   Y[2027] := 0.748582;
   Y[2028] := 0.7531839;
   Y[2029] := 0.7531839;
   Y[2030] := 0.75165;
   Y[2031] := 0.7531839;
   Y[2032] := 0.750116;
   Y[2033] := 0.7547179;
   Y[2034] := 0.748582;
   Y[2035] := 0.7593198;
   Y[2036] := 0.750116;
   Y[2037] := 0.7577859;
   Y[2038] := 0.7531839;
   Y[2039] := 0.7531839;
   Y[2040] := 0.745514;
   Y[2041] := 0.7639218;
   Y[2042] := 0.748582;
   Y[2043] := 0.7623878;
   Y[2044] := 0.750116;
   Y[2045] := 0.7577859;
   Y[2046] := 0.747048;
   Y[2047] := 0.7623878;
   Y[2048] := 0.748582;
   Y[2049] := 0.7700577;
   Y[2050] := 0.7424461;
   Y[2051] := 0.7608538;
   Y[2052] := 0.7531839;
   Y[2053] := 0.7577859;
   Y[2054] := 0.7531839;
   Y[2055] := 0.7577859;
   Y[2056] := 0.7577859;
   Y[2057] := 0.7531839;
   Y[2058] := 0.7593198;
   Y[2059] := 0.7531839;
   Y[2060] := 0.7623878;
   Y[2061] := 0.750116;
   Y[2062] := 0.7623878;
   Y[2063] := 0.7531839;
   Y[2064] := 0.7623878;
   Y[2065] := 0.750116;
   Y[2066] := 0.7654558;
   Y[2067] := 0.7562519;
   Y[2068] := 0.7577859;
   Y[2069] := 0.750116;
   Y[2070] := 0.7669898;
   Y[2071] := 0.747048;
   Y[2072] := 0.7669898;
   Y[2073] := 0.748582;
   Y[2074] := 0.7731256;
   Y[2075] := 0.747048;
   Y[2076] := 0.7654558;
   Y[2077] := 0.748582;
   Y[2078] := 0.7654558;
   Y[2079] := 0.750116;
   Y[2080] := 0.7608538;
   Y[2081] := 0.7547179;
   Y[2082] := 0.7562519;
   Y[2083] := 0.7562519;
   Y[2084] := 0.75165;
   Y[2085] := 0.7562519;
   Y[2086] := 0.7439801;
   Y[2087] := 0.7378441;
   Y[2088] := 0.7056305;
   Y[2089] := 0.6626791;
   Y[2090] := 0.5798442;
   Y[2091] := 0.523087;
   Y[2092] := 0.4617278;
   Y[2093] := 0.4203104;
   Y[2094] := 0.4003687;
   Y[2095] := 0.3926988;
   Y[2096] := 0.374291;
   Y[2097] := 0.3666211;
   Y[2098] := 0.3620192;
   Y[2099] := 0.3574172;
   Y[2100] := 0.3589512;
   Y[2101] := 0.3620192;
   Y[2102] := 0.3666211;
   Y[2103] := 0.3681551;
   Y[2104] := 0.3635531;
   Y[2105] := 0.3574172;
   Y[2106] := 0.3604852;
   Y[2107] := 0.3497473;
   Y[2108] := 0.3574172;
   Y[2109] := 0.3512813;
   Y[2110] := 0.3512813;
   Y[2111] := 0.3620192;
   Y[2112] := 0.3574172;
   Y[2113] := 0.3482133;
   Y[2114] := 0.3482133;
   Y[2115] := 0.3543493;
   Y[2116] := 0.3451454;
   Y[2117] := 0.3543493;
   Y[2118] := 0.3405434;
   Y[2119] := 0.3543493;
   Y[2120] := 0.3451454;
   Y[2121] := 0.3558832;
   Y[2122] := 0.3451454;
   Y[2123] := 0.3558832;
   Y[2124] := 0.3482133;
   Y[2125] := 0.3604852;
   Y[2126] := 0.3666211;
   Y[2127] := 0.3558832;
   Y[2128] := 0.3650871;
   Y[2129] := 0.3589512;
   Y[2130] := 0.3620192;
   Y[2131] := 0.3466794;
   Y[2132] := 0.3497473;
   Y[2133] := 0.3574172;
   Y[2134] := 0.3589512;
   Y[2135] := 0.369689;
   Y[2136] := 0.3635531;
   Y[2137] := 0.3788929;
   Y[2138] := 0.369689;
   Y[2139] := 0.3773589;
   Y[2140] := 0.372757;
   Y[2141] := 0.371223;
   Y[2142] := 0.3819609;
   Y[2143] := 0.375825;
   Y[2144] := 0.3773589;
   Y[2145] := 0.372757;
   Y[2146] := 0.3911648;
   Y[2147] := 0.3880968;
   Y[2148] := 0.371223;
   Y[2149] := 0.374291;
   Y[2150] := 0.374291;
   Y[2151] := 0.374291;
   Y[2152] := 0.374291;
   Y[2153] := 0.3681551;
   Y[2154] := 0.3788929;
   Y[2155] := 0.3804269;
   Y[2156] := 0.3834949;
   Y[2157] := 0.3865628;
   Y[2158] := 0.3926988;
   Y[2159] := 0.3926988;
   Y[2160] := 0.3865628;
   Y[2161] := 0.3942327;
   Y[2162] := 0.3804269;
   Y[2163] := 0.3911648;
   Y[2164] := 0.3880968;
   Y[2165] := 0.3880968;
   Y[2166] := 0.3865628;
   Y[2167] := 0.3988347;
   Y[2168] := 0.3942327;
   Y[2169] := 0.3819609;
   Y[2170] := 0.3911648;
   Y[2171] := 0.3988347;
   Y[2172] := 0.3911648;
   Y[2173] := 0.3850288;
   Y[2174] := 0.4003687;
   Y[2175] := 0.3926988;
   Y[2176] := 0.3896308;
   Y[2177] := 0.369689;
   Y[2178] := 0.3788929;
   Y[2179] := 0.3834949;
   Y[2180] := 0.3973007;
   Y[2181] := 0.3850288;
   Y[2182] := 0.3957667;
   Y[2183] := 0.3911648;
   Y[2184] := 0.4049706;
   Y[2185] := 0.3957667;
   Y[2186] := 0.4111065;
   Y[2187] := 0.4126405;
   Y[2188] := 0.4049706;
   Y[2189] := 0.4034366;
   Y[2190] := 0.4157085;
   Y[2191] := 0.4187764;
   Y[2192] := 0.4126405;
   Y[2193] := 0.4203104;
   Y[2194] := 0.4187764;
   Y[2195] := 0.4264463;
   Y[2196] := 0.4095725;
   Y[2197] := 0.4279803;
   Y[2198] := 0.4172424;
   Y[2199] := 0.4325822;
   Y[2200] := 0.4141745;
   Y[2201] := 0.4341162;
   Y[2202] := 0.4325822;
   Y[2203] := 0.4325822;
   Y[2204] := 0.4233783;
   Y[2205] := 0.4295143;
   Y[2206] := 0.4448541;
   Y[2207] := 0.4295143;
   Y[2208] := 0.4264463;
   Y[2209] := 0.4249123;
   Y[2210] := 0.4371842;
   Y[2211] := 0.4203104;
   Y[2212] := 0.4233783;
   Y[2213] := 0.4249123;
   Y[2214] := 0.4264463;
   Y[2215] := 0.4141745;
   Y[2216] := 0.4187764;
   Y[2217] := 0.4295143;
   Y[2218] := 0.4295143;
   Y[2219] := 0.4203104;
   Y[2220] := 0.4264463;
   Y[2221] := 0.4249123;
   Y[2222] := 0.4203104;
   Y[2223] := 0.4111065;
   Y[2224] := 0.4157085;
   Y[2225] := 0.4264463;
   Y[2226] := 0.4065046;
   Y[2227] := 0.4141745;
   Y[2228] := 0.4218444;
   Y[2229] := 0.4310482;
   Y[2230] := 0.4187764;
   Y[2231] := 0.4218444;
   Y[2232] := 0.4264463;
   Y[2233] := 0.4233783;
   Y[2234] := 0.4203104;
   Y[2235] := 0.4310482;
   Y[2236] := 0.4341162;
   Y[2237] := 0.4203104;
   Y[2238] := 0.4187764;
   Y[2239] := 0.4218444;
   Y[2240] := 0.4295143;
   Y[2241] := 0.4141745;
   Y[2242] := 0.4203104;
   Y[2243] := 0.4203104;
   Y[2244] := 0.4233783;
   Y[2245] := 0.4126405;
   Y[2246] := 0.4233783;
   Y[2247] := 0.4310482;
   Y[2248] := 0.4279803;
   Y[2249] := 0.4279803;
   Y[2250] := 0.4295143;
   Y[2251] := 0.4310482;
   Y[2252] := 0.4249123;
   Y[2253] := 0.4264463;
   Y[2254] := 0.4295143;
   Y[2255] := 0.4264463;
   Y[2256] := 0.4264463;
   Y[2257] := 0.4341162;
   Y[2258] := 0.4356502;
   Y[2259] := 0.4325822;
   Y[2260] := 0.4402521;
   Y[2261] := 0.4571259;
   Y[2262] := 0.4540579;
   Y[2263] := 0.4387181;
   Y[2264] := 0.4540579;
   Y[2265] := 0.4632618;
   Y[2266] := 0.4571259;
   Y[2267] := 0.446388;
   Y[2268] := 0.4525239;
   Y[2269] := 0.4402521;
   Y[2270] := 0.4402521;
   Y[2271] := 0.4371842;
   Y[2272] := 0.4555919;
   Y[2273] := 0.4387181;
   Y[2274] := 0.4433201;
   Y[2275] := 0.4448541;
   Y[2276] := 0.4555919;
   Y[2277] := 0.4371842;
   Y[2278] := 0.4448541;
   Y[2279] := 0.449456;
   Y[2280] := 0.4433201;
   Y[2281] := 0.4325822;
   Y[2282] := 0.4371842;
   Y[2283] := 0.4356502;
   Y[2284] := 0.4187764;
   Y[2285] := 0.4203104;
   Y[2286] := 0.4187764;
   Y[2287] := 0.4095725;
   Y[2288] := 0.4126405;
   Y[2289] := 0.4233783;
   Y[2290] := 0.4279803;
   Y[2291] := 0.4157085;
   Y[2292] := 0.4080386;
   Y[2293] := 0.3957667;
   Y[2294] := 0.4003687;
   Y[2295] := 0.3773589;
   Y[2296] := 0.374291;
   Y[2297] := 0.3896308;
   Y[2298] := 0.3880968;
   Y[2299] := 0.3804269;
   Y[2300] := 0.371223;
   Y[2301] := 0.3788929;
   Y[2302] := 0.3804269;
   Y[2303] := 0.3451454;
   Y[2304] := 0.3604852;
   Y[2305] := 0.3650871;
   Y[2306] := 0.3589512;
   Y[2307] := 0.3390095;
   Y[2308] := 0.3267376;
   Y[2309] := 0.3451454;
   Y[2310] := 0.3344075;
   Y[2311] := 0.3374755;
   Y[2312] := 0.3083299;
   Y[2313] := 0.2883881;
   Y[2314] := 0.2899221;
   Y[2315] := 0.2807182;
   Y[2316] := 0.2822522;
   Y[2317] := 0.2669124;
   Y[2318] := 0.2607765;
   Y[2319] := 0.2500387;
   Y[2320] := 0.2515726;
   Y[2321] := 0.2454367;
   Y[2322] := 0.2715144;
   Y[2323] := 0.2653784;
   Y[2324] := 0.2377668;
   Y[2325] := 0.228563;
   Y[2326] := 0.2393008;
   Y[2327] := 0.2592425;
   Y[2328] := 0.2669124;
   Y[2329] := 0.2899221;
   Y[2330] := 0.2745823;
   Y[2331] := 0.2592425;
   Y[2332] := 0.2883881;
   Y[2333] := 0.2715144;
   Y[2334] := 0.2761163;
   Y[2335] := 0.2745823;
   Y[2336] := 0.2653784;
   Y[2337] := 0.2577085;
   Y[2338] := 0.2546406;
   Y[2339] := 0.2454367;
   Y[2340] := 0.2439027;
   Y[2341] := 0.2423688;
   Y[2342] := 0.2377668;
   Y[2343] := 0.2316309;
   Y[2344] := 0.220893;
   Y[2345] := 0.2178251;
   Y[2346] := 0.2132231;
   Y[2347] := 0.2147571;
   Y[2348] := 0.2086212;
   Y[2349] := 0.2086212;
   Y[2350] := 0.1994173;
   Y[2351] := 0.1917474;
   Y[2352] := 0.1902135;
   Y[2353] := 0.1856115;
   Y[2354] := 0.1810096;
   Y[2355] := 0.1810096;
   Y[2356] := 0.1794756;
   Y[2357] := 0.1764076;
   Y[2358] := 0.1718057;
   Y[2359] := 0.1656698;
   Y[2360] := 0.1610678;
   Y[2361] := 0.1579999;
   Y[2362] := 0.1564659;
   Y[2363] := 0.15033;
   Y[2364] := 0.148796;
   Y[2365] := 0.148796;
   Y[2366] := 0.147262;
   Y[2367] := 0.1457281;
   Y[2368] := 0.1411261;
   Y[2369] := 0.1380582;
   Y[2370] := 0.1334562;
   Y[2371] := 0.1303883;
   Y[2372] := 0.1273203;
   Y[2373] := 0.1257863;
   Y[2374] := 0.1211844;
   Y[2375] := 0.1196504;
   Y[2376] := 0.1181164;
   Y[2377] := 0.1181164;
   Y[2378] := 0.1165824;
   Y[2379] := 0.1150485;
   Y[2380] := 0.1135145;
   Y[2381] := 0.1089125;
   Y[2382] := 0.1073786;
   Y[2383] := 0.1043106;
   Y[2384] := 0.1012426;
   Y[2385] := 0.1012426;
   Y[2386] := 0.09664071;
   Y[2387] := 0.09664071;
   Y[2388] := 0.09357275;
   Y[2389] := 0.09357275;
   Y[2390] := 0.09050479;
   Y[2391] := 0.08897081;
   Y[2392] := 0.08897081;
   Y[2393] := 0.08897081;
   Y[2394] := 0.08743683;
   Y[2395] := 0.08743683;
   Y[2396] := 0.08436887;
   Y[2397] := 0.08283489;
   Y[2398] := 0.08130091;
   Y[2399] := 0.07976694;
   Y[2400] := 0.07823295;
   Y[2401] := 0.075165;
   Y[2402] := 0.07363102;
   Y[2403] := 0.07363102;
   Y[2404] := 0.07209703;
   Y[2405] := 0.07056306;
   Y[2406] := 0.06902908;
   Y[2407] := 0.06902908;
   Y[2408] := 0.0674951;
   Y[2409] := 0.06596112;
   Y[2410] := 0.06596112;
   Y[2411] := 0.06289316;
   Y[2412] := 0.06442714;
   Y[2413] := 0.06289316;
   Y[2414] := 0.06289316;
   Y[2415] := 0.06135918;
   Y[2416] := 0.06135918;
   Y[2417] := 0.06135918;
   Y[2418] := 0.0598252;
   Y[2419] := 0.0598252;
   Y[2420] := 0.0598252;
   Y[2421] := 0.05829122;
   Y[2422] := 0.05675724;
   Y[2423] := 0.05522326;
   Y[2424] := 0.05368928;
   Y[2425] := 0.0521553;
   Y[2426] := 0.0521553;
   Y[2427] := 0.05062132;
   Y[2428] := 0.05062132;
   Y[2429] := 0.05062132;
   Y[2430] := 0.05062132;
   Y[2431] := 0.04755336;
   Y[2432] := 0.04908735;
   Y[2433] := 0.04601939;
   Y[2434] := 0.04755336;
   Y[2435] := 0.04601939;
   Y[2436] := 0.04601939;
   Y[2437] := 0.04601939;
   Y[2438] := 0.04295143;
   Y[2439] := 0.04295143;
   Y[2440] := 0.04295143;
   Y[2441] := 0.04141745;
   Y[2442] := 0.04141745;
   Y[2443] := 0.04141745;
   Y[2444] := 0.04295143;
   Y[2445] := 0.04141745;
   Y[2446] := 0.04141745;
   Y[2447] := 0.03988347;
   Y[2448] := 0.03988347;
   Y[2449] := 0.03988347;
   Y[2450] := 0.04141745;
   Y[2451] := 0.03988347;
   Y[2452] := 0.03988347;
   Y[2453] := 0.03988347;
   Y[2454] := 0.03988347;
   Y[2455] := 0.03834949;
   Y[2456] := 0.03988347;
   Y[2457] := 0.03681551;
   Y[2458] := 0.03681551;
   Y[2459] := 0.03681551;
   Y[2460] := 0.03374755;
   Y[2461] := 0.03528153;
   Y[2462] := 0.03374755;
   Y[2463] := 0.03221357;
   Y[2464] := 0.03374755;
   Y[2465] := 0.03374755;
   Y[2466] := 0.03221357;
   Y[2467] := 0.03528153;
   Y[2468] := 0.03374755;
   Y[2469] := 0.03221357;
   Y[2470] := 0.03374755;
   Y[2471] := 0.03221357;
   Y[2472] := 0.03374755;
   Y[2473] := 0.03221357;
   Y[2474] := 0.03221357;
   Y[2475] := 0.03221357;
   Y[2476] := 0.03221357;
   Y[2477] := 0.03221357;
   Y[2478] := 0.03067959;
   Y[2479] := 0.03067959;
   Y[2480] := 0.03067959;
   Y[2481] := 0.02914561;
   Y[2482] := 0.02914561;
   Y[2483] := 0.02761163;
   Y[2484] := 0.02914561;
   Y[2485] := 0.02607765;
   Y[2486] := 0.02761163;
   Y[2487] := 0.02761163;
   Y[2488] := 0.02761163;
   Y[2489] := 0.02761163;
   Y[2490] := 0.02761163;
   Y[2491] := 0.02914561;
   Y[2492] := 0.02761163;
   Y[2493] := 0.02914561;
   Y[2494] := 0.02761163;
   Y[2495] := 0.02761163;
   Y[2496] := 0.02761163;
   Y[2497] := 0.02607765;
   Y[2498] := 0.02914561;
   Y[2499] := 0.02761163;

END_DATA_BLOCK

FUNCTION "VecDivVal" : Void
{ S7_Optimized_Access := 'TRUE' }
VERSION : 0.1
   VAR_INPUT
      A : Array[0.."n"] of Real;
      val : Real;
   END_VAR

   VAR_OUTPUT
      C : Array[0.."n"] of Real;
   END_VAR

   VAR_TEMP
      i : DInt;
      j : DInt;
   END_VAR


BEGIN
	FOR #i := 0 TO "n" DO
	    #C[#i] := #A[#i] / #val;
	END_FOR;

END_FUNCTION

FUNCTION "MulVecRowVecCol" : Void
{ S7_Optimized_Access := 'TRUE' }
VERSION : 0.1
   VAR_INPUT
      A : Array[0.."n"] of Real;
      B : Array[0.."n"] of Real;
   END_VAR

   VAR_OUTPUT
      s : Real;
   END_VAR

   VAR_TEMP
      i : DInt;
   END_VAR


BEGIN
	#s := 0.0;
	FOR #i := 0 TO "n" DO
	    #s := #s + #A[#i] * #B[#i];
	END_FOR;

END_FUNCTION

FUNCTION "MulVecColVecRow" : Void
{ S7_Optimized_Access := 'TRUE' }
VERSION : 0.1
   VAR_INPUT
      A : Array[0.."n"] of Real;
      B : Array[0.."n"] of Real;
   END_VAR

   VAR_OUTPUT
      C : Array[0.."n", 0.."n"] of Real;
   END_VAR

   VAR_TEMP
      i : DInt;
      j : DInt;
   END_VAR


BEGIN
	FOR #i := 0 TO "n" DO
	    FOR #j := 0 TO "n" DO
	        #C[#i, #j] := #A[#i] * #B[#j];
	    END_FOR;
	END_FOR;

END_FUNCTION

FUNCTION "MulMatVecCol" : Void
{ S7_Optimized_Access := 'TRUE' }
VERSION : 0.1
   VAR_INPUT
      A : Array[0.."n", 0.."n"] of Real;
      B : Array[0.."n"] of Real;
   END_VAR

   VAR_OUTPUT
      C : Array[0.."n"] of Real;
   END_VAR

   VAR_TEMP
      i : DInt;
      j : DInt;
      k : DInt;
   END_VAR


BEGIN
	"VecFilled"(val := 0.0,
	            C => #C);

	FOR #i := 0 TO "n" DO
	    FOR #j := 0 TO "n" DO
	        #C[#i] := #C[#i] + #A[#i, #j] * #B[#j];
	    END_FOR;
	END_FOR;

END_FUNCTION

DATA_BLOCK "Scheduler"
{ S7_Optimized_Access := 'TRUE' }
VERSION : 0.1
NON_RETAIN
   VAR
      tm_break : Bool;
      flag_global : UDInt;
      flag_iter : UDInt;
      time_start {InstructionName := 'DTL'; LibVersion := '1.0'} : DTL;
      time_bound : UDInt;   // 50ms
      time_check {InstructionName := 'DTL'; LibVersion := '1.0'} : DTL;
      time_duration : UDInt;
   END_VAR


BEGIN
   time_bound := 50000000;

END_DATA_BLOCK

FUNCTION "MatDivVal" : Void
{ S7_Optimized_Access := 'TRUE' }
VERSION : 0.1
   VAR_INPUT
      A : Array[0.."n", 0.."n"] of Real;
      val : Real;
   END_VAR

   VAR_OUTPUT
      C : Array[0.."n", 0.."n"] of Real;
   END_VAR

   VAR_TEMP
      i : DInt;
      j : DInt;
   END_VAR


BEGIN
	FOR #i := 0 TO "n" DO
	    FOR #j := 0 TO "n" DO
	        #C[#i, #j] := #A[#i, #j] / #val;
	    END_FOR;
	END_FOR;

END_FUNCTION

FUNCTION "MulMatMat" : Void
{ S7_Optimized_Access := 'TRUE' }
VERSION : 0.1
   VAR_INPUT
      A : Array[0.."n", 0.."n"] of Real;
      B : Array[0.."n", 0.."n"] of Real;
   END_VAR

   VAR_OUTPUT
      C : Array[0.."n", 0.."n"] of Real;
   END_VAR

   VAR_TEMP
      i : DInt;
      j : DInt;
      k : DInt;
   END_VAR


BEGIN
	"MatFilled"(val := 0,
	            C => #C);

	FOR #i := 0 TO "n" DO
	    FOR #j := 0 TO "n" DO
	        FOR #k := 0 TO "n" DO
	            #C[#i, #j] := #C[#i, #j] + #A[#i, #k] * #B[#k, #j];
	        END_FOR;
	    END_FOR;
	END_FOR;

END_FUNCTION

FUNCTION "EwrlsSetEps" : Void
{ S7_Optimized_Access := 'TRUE' }
VERSION : 0.1
   VAR_INPUT
      Phi : Array[0.."n"] of Real;
      Theta : Array[0.."n"] of Real;
   END_VAR

   VAR_IN_OUT
      eps : Real;
   END_VAR

   VAR_TEMP
      j : DInt;
      status : Int;
   END_VAR


BEGIN
	//if there is no break or this is the correct function
	IF (NOT "Scheduler".tm_break) OR ("Scheduler".tm_break AND "Scheduler".flag_iter = "Scheduler".flag_global) THEN
	    //correct function -> cancel the break
	    IF "Scheduler".tm_break THEN
	        "Scheduler".tm_break := FALSE;
	    END_IF;

	    //local flag = global flag
	    "Scheduler".flag_iter := "Scheduler".flag_global;

	    //time check
	    #status := RD_LOC_T("Scheduler".time_check);
	    IF "Scheduler".time_check.SECOND = "Scheduler".time_start.SECOND + 1 THEN
	        "Scheduler".time_duration := 1_000_000_000 + "Scheduler".time_check.NANOSECOND - "Scheduler".time_start.NANOSECOND;
	    ELSIF "Scheduler".time_check.SECOND = "Scheduler".time_start.SECOND THEN
	        "Scheduler".time_duration := "Scheduler".time_check.NANOSECOND - "Scheduler".time_start.NANOSECOND;
	    END_IF;

	    //if computation time is too long then make a break
	    IF "Scheduler".time_duration > "Scheduler".time_bound THEN
	        "Scheduler".tm_break := TRUE;
	        RETURN;
	    ELSE
	        // Calculate residual error: eps(i) = y(i) - Phi(i)' * Theta(i-1)
	        #eps := "Db_1".Y["i"];
	        FOR #j := 0 TO "n" DO
	            #eps := #eps - #Phi[#j] * #Theta[#j];
	        END_FOR;
	    END_IF;
	    //iterate global flag
	    "Scheduler".flag_global := "Scheduler".flag_global + 1;
	END_IF;

END_FUNCTION

FUNCTION "EwrlsSetTheta" : Void
{ S7_Optimized_Access := 'TRUE' }
VERSION : 0.1
   VAR_INPUT
      K : Array[0.."n"] of Real;
      eps : Real;
   END_VAR

   VAR_IN_OUT
      Theta : Array[0.."n"] of Real;
   END_VAR

   VAR_TEMP
      j : DInt;
      status : Int;
   END_VAR


BEGIN
	//if there is no break or this is the correct function
	IF (NOT "Scheduler".tm_break) OR ("Scheduler".tm_break AND "Scheduler".flag_iter = "Scheduler".flag_global) THEN
	    //correct function -> cancel the break
	    IF "Scheduler".tm_break THEN
	        "Scheduler".tm_break := FALSE;
	    END_IF;

	    //local flag = global flag
	    "Scheduler".flag_iter := "Scheduler".flag_global;

	    //time check
	    #status := RD_LOC_T("Scheduler".time_check);
	    IF "Scheduler".time_check.SECOND = "Scheduler".time_start.SECOND + 1 THEN
	        "Scheduler".time_duration := 1_000_000_000 + "Scheduler".time_check.NANOSECOND - "Scheduler".time_start.NANOSECOND;
	    ELSIF "Scheduler".time_check.SECOND = "Scheduler".time_start.SECOND THEN
	        "Scheduler".time_duration := "Scheduler".time_check.NANOSECOND - "Scheduler".time_start.NANOSECOND;
	    END_IF;

	    //if computation time is too long then make a break
	    IF "Scheduler".time_duration > "Scheduler".time_bound THEN
	        "Scheduler".tm_break := TRUE;
	        RETURN;
	    ELSE
	        // Calculate parameter vector: Theta(i) = Theta(i-1) + K(i) * eps(i)
	        FOR #j := 0 TO "n" DO
	            #Theta[#j] := #Theta[#j] + #K[#j] * #eps;
	        END_FOR;
	    END_IF;
	    //iterate global flag
	    "Scheduler".flag_global := "Scheduler".flag_global + 1;
	END_IF;

END_FUNCTION

FUNCTION "EwrlsSetK" : Void
{ S7_Optimized_Access := 'TRUE' }
VERSION : 0.1
   VAR_INPUT
      P : Array[0.."n", 0.."n"] of Real;
      Phi : Array[0.."n"] of Real;
      lambda : Real;
   END_VAR

   VAR_IN_OUT
      K : Array[0.."n"] of Real;
   END_VAR

   VAR_TEMP
      Vec1 : Array[0.."n"] of Real;
      div : Real;
      status : Int;
   END_VAR


BEGIN
	//if there is no break or this is the correct function
	IF (NOT "Scheduler".tm_break) OR ("Scheduler".tm_break AND "Scheduler".flag_iter = "Scheduler".flag_global) THEN
	    //correct function -> cancel the break
	    IF "Scheduler".tm_break THEN
	        "Scheduler".tm_break := FALSE;
	    END_IF;

	    //local flag = global flag
	    "Scheduler".flag_iter := "Scheduler".flag_global;

	    //time check
	    #status := RD_LOC_T("Scheduler".time_check);
	    IF "Scheduler".time_check.SECOND = "Scheduler".time_start.SECOND + 1 THEN
	        "Scheduler".time_duration := 1_000_000_000 + "Scheduler".time_check.NANOSECOND - "Scheduler".time_start.NANOSECOND;
	    ELSIF "Scheduler".time_check.SECOND = "Scheduler".time_start.SECOND THEN
	        "Scheduler".time_duration := "Scheduler".time_check.NANOSECOND - "Scheduler".time_start.NANOSECOND;
	    END_IF;

	    //if computation time is too long then make a break
	    IF "Scheduler".time_duration > "Scheduler".time_bound THEN
	        "Scheduler".tm_break := TRUE;
	        RETURN;
	    ELSE
	        // Calculate K: K(i) = (P(i-1) * Phi(i)) / (lambda + Phi(i)' * P(i-1) * Phi(i))
	        "MulMatVecCol"(A := #P,
	                       B := #Phi,
	                       C => #Vec1);
	        "MulVecRowVecCol"(A := #Phi,
	                          B := #Vec1,
	                          s => #div);
	        #div := #div + #lambda;
	        "VecDivVal"(A := #Vec1,
	                    val := #div,
	                    C => #K);
	    END_IF;
	    //iterate global flag
	    "Scheduler".flag_global := "Scheduler".flag_global + 1;
	END_IF;

END_FUNCTION

FUNCTION "EwrlsSetPhi" : Void
{ S7_Optimized_Access := 'TRUE' }
VERSION : 0.1
   VAR_OUTPUT
      Phi : Array[0.."n"] of Real;
   END_VAR

   VAR_TEMP
      j : DInt;
      status : Int;
   END_VAR


BEGIN
	//if there is no break or this is the correct function
	IF (NOT "Scheduler".tm_break) OR ("Scheduler".tm_break AND "Scheduler".flag_iter = "Scheduler".flag_global) THEN
	    //correct function -> cancel the break
	    IF "Scheduler".tm_break THEN
	        "Scheduler".tm_break := FALSE;
	    END_IF;

	    //local flag = global flag
	    "Scheduler".flag_iter := "Scheduler".flag_global;

	    //time check
	    #status := RD_LOC_T("Scheduler".time_check);
	    IF "Scheduler".time_check.SECOND = "Scheduler".time_start.SECOND + 1 THEN
	        "Scheduler".time_duration := 1_000_000_000 + "Scheduler".time_check.NANOSECOND - "Scheduler".time_start.NANOSECOND;
	    ELSIF "Scheduler".time_check.SECOND = "Scheduler".time_start.SECOND THEN
	        "Scheduler".time_duration := "Scheduler".time_check.NANOSECOND - "Scheduler".time_start.NANOSECOND;
	    END_IF;

	    //if computation time is too long then make a break
	    IF "Scheduler".time_duration > "Scheduler".time_bound THEN
	        "Scheduler".tm_break := TRUE;
	        RETURN;
	    ELSE
	        // Set values inside regression vector: Phi(i) = [y(i-1) ... y(i-a+1) u(i-1) ... u(i-b+1)]
	        FOR #j := 0 TO "a" - 1 DO
	            #Phi[#j] := "Db_1".Y["i" - #j - 1];
	        END_FOR;
	        FOR #j := "a" TO "n" DO
	            #Phi[#j] := "Db_1".U["i" + "a" - #j - 1];
	        END_FOR;
	    END_IF;
	    //iterate global flag
	    "Scheduler".flag_global := "Scheduler".flag_global + 1;
	END_IF;

END_FUNCTION

FUNCTION "EwrlsSetP" : Void
{ S7_Optimized_Access := 'TRUE' }
VERSION : 0.1
   VAR_INPUT
      K : Array[0.."n"] of Real;
      Phi : Array[0.."n"] of Real;
      lambda : Real;
   END_VAR

   VAR_IN_OUT
      P : Array[0.."n", 0.."n"] of Real;
   END_VAR

   VAR_TEMP
      Mat1 : Array[0.."n", 0.."n"] of Real;
      Mat2 : Array[0.."n", 0.."n"] of Real;
      Mat3 : Array[0.."n", 0.."n"] of Real;
      status : Int;
   END_VAR


BEGIN
	//if there is no break or this is the correct function
	IF (NOT "Scheduler".tm_break) OR ("Scheduler".tm_break AND "Scheduler".flag_iter = "Scheduler".flag_global) THEN
	    //correct function -> cancel the break
	    IF "Scheduler".tm_break THEN
	        "Scheduler".tm_break := FALSE;
	    END_IF;

	    //local flag = global flag
	    "Scheduler".flag_iter := "Scheduler".flag_global;

	    //time check
	    #status := RD_LOC_T("Scheduler".time_check);
	    IF "Scheduler".time_check.SECOND = "Scheduler".time_start.SECOND + 1 THEN
	        "Scheduler".time_duration := 1_000_000_000 + "Scheduler".time_check.NANOSECOND - "Scheduler".time_start.NANOSECOND;
	    ELSIF "Scheduler".time_check.SECOND = "Scheduler".time_start.SECOND THEN
	        "Scheduler".time_duration := "Scheduler".time_check.NANOSECOND - "Scheduler".time_start.NANOSECOND;
	    END_IF;

	    //if computation time is too long then make a break
	    IF "Scheduler".time_duration > "Scheduler".time_bound THEN
	        "Scheduler".tm_break := TRUE;
	        RETURN;
	    ELSE
	        // Calculate P: P(i) = (P(i-1) - K(i) * Phi(i)' * P(i-1)) / lambda
	        "MulVecColVecRow"(A := #K,
	                          B := #Phi,
	                          C => #Mat1);
	        "MulMatMat"(A := #Mat1,
	                    B := #P,
	                    C => #Mat2);
	        "SubMatMat"(A := #P,
	                    B := #Mat2,
	                    C => #Mat3);
	        "MatDivVal"(A := #Mat3,
	                    val := #lambda,
	                    C => #P);
	    END_IF;
	    //iterate global flag
	    "Scheduler".flag_global := "Scheduler".flag_global + 1;
	END_IF;

END_FUNCTION

FUNCTION_BLOCK "ewrls"
{ S7_Optimized_Access := 'TRUE' }
VERSION : 0.1
   VAR
      eps : Real;
      Phi : Array[0.."n"] of Real;
      K : Array[0.."n"] of Real;
      P : Array[0.."n", 0.."n"] of Real;
      Theta : Array[0.."n"] of Real;
      lambda : Real;
   END_VAR

   VAR_TEMP
      j : DInt;
      div : Real;
      Vec1 : Array[0.."n"] of Real;
      Mat1 : Array[0.."n", 0.."n"] of Real;
      Mat2 : Array[0.."n", 0.."n"] of Real;
      Mat3 : Array[0.."n", 0.."n"] of Real;
   END_VAR


BEGIN
	// At the end, the coefficients will be in "Db_1".Theta
	// does approx 117-118 iterations per default cycle (not scheduled)
	WHILE "i" <= "M" DO
	    // Set values inside regression vector: Phi(i) = [y(i-1) ... y(i-a+1) u(i-1) ... u(i-b+1)]
	    "EwrlsSetPhi"(Phi => #Phi);
	    // Calculate residual error: eps(i) = y(i) - Phi(i)' * Theta(i-1)
	    "EwrlsSetEps"(Phi := #Phi,
	                  Theta := #Theta,
	                  eps := #eps);
	    // Calculate K: K(i) = (P(i-1) * Phi(i)) / (lambda + Phi(i)' * P(i-1) * Phi(i))
	    "EwrlsSetK"(P := #P,
	                Phi := #Phi,
	                lambda := #lambda,
	                K := #K);
	    // Calculate parameter vector: Theta(i) = Theta(i-1) + K(i) * eps(i)
	    "EwrlsSetTheta"(K := #K,
	                    eps := #eps,
	                    Theta := #Theta);
	    // Calculate P: P(i) = (P(i-1) - K(i) * Phi(i)' * P(i-1)) / lambda
	    "EwrlsSetP"(K := #K,
	                Phi := #Phi,
	                lambda := #lambda,
	                P := #P);
	    IF NOT "Scheduler".tm_break THEN
	        "i" := "i" + 1;
	    ELSE
	        EXIT;
	    END_IF;
	END_WHILE;

END_FUNCTION_BLOCK

DATA_BLOCK "ewrls_DB"
{ S7_Optimized_Access := 'TRUE' }
VERSION : 0.1
NON_RETAIN
"ewrls"

BEGIN

END_DATA_BLOCK

FUNCTION "MatIdentity" : Void
{ S7_Optimized_Access := 'TRUE' }
VERSION : 0.1
   VAR_INPUT
      val : Real;
   END_VAR

   VAR_OUTPUT
      C : Array[0.."n", 0.."n"] of Real;
   END_VAR

   VAR_TEMP
      i : DInt;
   END_VAR


BEGIN
	"MatFilled"(val := 0.0,
	            C => #C);
	FOR #i := 0 TO "n" DO
	    #C[#i, #i] := #val;
	END_FOR;

END_FUNCTION

FUNCTION_BLOCK "calculate_mse"
{ S7_Optimized_Access := 'TRUE' }
VERSION : 0.1

BEGIN
	"mean_squared_error" := "mean_squared_error" / DINT_TO_LREAL("M" + 1);

END_FUNCTION_BLOCK

FUNCTION_BLOCK "ewrls_initialization"
{ S7_Optimized_Access := 'TRUE' }
VERSION : 0.1
   VAR_TEMP
      c : Real;
   END_VAR


BEGIN
	"ewrls_DB".lambda := 1.00; // forgetting factor (=1 means no forgetting)
	#c := 1_000_000; //"large number" to initialize P
	"MatIdentity"(val := #c,
	              C => "ewrls_DB".P);
	// Pad input and output vectors with "n" zeros at the beginning
	"i" := MAX(IN1 := "a", IN2 := "b");
	"VecFilled"(val := 0.0,
	            C => "ewrls_DB".Theta);
	"mean_squared_error" := 0.0;
	"initEwrls" := FALSE;

END_FUNCTION_BLOCK

FUNCTION_BLOCK "mse"
{ S7_Optimized_Access := 'TRUE' }
VERSION : 0.1
   VAR_TEMP
      iter_error : LReal;
      j : DInt;
      status : Int;
   END_VAR


BEGIN
	WHILE "i" <= "M" DO
	    //if there is no break or this is the correct function
	    IF (NOT "Scheduler".tm_break) OR ("Scheduler".tm_break AND "Scheduler".flag_iter = "Scheduler".flag_global) THEN
	        //correct function -> cancel the break
	        IF "Scheduler".tm_break THEN
	            "Scheduler".tm_break := FALSE;
	        END_IF;

	        //local flag = global flag
	        "Scheduler".flag_iter := "Scheduler".flag_global;

	        //time check
	        #status := RD_LOC_T("Scheduler".time_check);
	        IF "Scheduler".time_check.SECOND = "Scheduler".time_start.SECOND + 1 THEN
	            "Scheduler".time_duration := 1_000_000_000 + "Scheduler".time_check.NANOSECOND - "Scheduler".time_start.NANOSECOND;
	        ELSIF "Scheduler".time_check.SECOND = "Scheduler".time_start.SECOND THEN
	            "Scheduler".time_duration := "Scheduler".time_check.NANOSECOND - "Scheduler".time_start.NANOSECOND;
	        END_IF;

	        //if computation time is too long then make a break
	        IF "Scheduler".time_duration > "Scheduler".time_bound THEN
	            "Scheduler".tm_break := TRUE;
	        END_IF;

	        //if there is no break - compute normally
	        IF NOT "Scheduler".tm_break THEN
	            #iter_error := "Db_1".Y["i"];
	            FOR #j := 0 TO "a" - 1 DO
	                #iter_error := #iter_error - "ewrls_DB".Theta[#j] * "Db_1".Y["i" - #j - 1];
	            END_FOR;
	            FOR #j := "a" TO "n" DO
	                #iter_error := #iter_error - "ewrls_DB".Theta[#j] * "Db_1".U["i" + "a" - #j - 1];
	            END_FOR;
	            #iter_error := #iter_error * #iter_error;
	            "mean_squared_error" := "mean_squared_error" + #iter_error;
	        END_IF;
	    END_IF;

	    IF NOT "Scheduler".tm_break THEN
	        "i" := "i" + 1;
	    ELSE
	        EXIT;
	    END_IF;
	END_WHILE;

END_FUNCTION_BLOCK

FUNCTION_BLOCK "array_initialization"
{ S7_Optimized_Access := 'TRUE' }
VERSION : 0.1

BEGIN


	"initArrays" := FALSE;

END_FUNCTION_BLOCK

DATA_BLOCK "mse_DB"
{ S7_Optimized_Access := 'TRUE' }
VERSION : 0.1
NON_RETAIN
"mse"

BEGIN

END_DATA_BLOCK

DATA_BLOCK "array_initialization_DB"
{ S7_Optimized_Access := 'TRUE' }
VERSION : 0.1
NON_RETAIN
"array_initialization"

BEGIN

END_DATA_BLOCK

DATA_BLOCK "calculate_mse_DB"
{ S7_Optimized_Access := 'TRUE' }
VERSION : 0.1
NON_RETAIN
"calculate_mse"

BEGIN

END_DATA_BLOCK

FUNCTION "SchedulerInit" : Void
{ S7_Optimized_Access := 'TRUE' }
VERSION : 0.1
   VAR_TEMP
      status : Int;
   END_VAR


BEGIN
	#status := RD_LOC_T("Scheduler".time_start);
	// "Scheduler".flag_global := 0;

END_FUNCTION

DATA_BLOCK "ewrls_initialization_DB"
{ S7_Optimized_Access := 'TRUE' }
VERSION : 0.1
NON_RETAIN
"ewrls_initialization"

BEGIN

END_DATA_BLOCK

